FUNCTION_BLOCK A2X_OR_2 (* Composite FB to calculate boolean OR between 2 A2X adapters (UP and DOWN independently) *)
  (* Standard: 61499-2; Function: OUT.UP = IN1.UP OR IN2.UP, OUT.DOWN = IN1.DOWN OR IN2.DOWN; Description: Copyright (c) 2026 HR Agrartechnik GmbH This program and the accompanying materials are made available under the terms of the Eclipse Public License 2.0 which is available at https://www.eclipse.org/legal/epl-2.0/ SPDX-License-Identifier: EPL-2.0 *)
  (* Version 1.0, 2026-08-31, Franz Höpfinger, HR Agrartechnik GmbH, Initial Version *)
  PACKAGE adapter::booleanOperators;
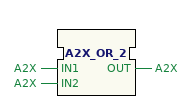
  SOCKETS
    IN1 : adapter::types::unidirectional::A2X; (* OR input 1 *)
    IN2 : adapter::types::unidirectional::A2X; (* OR input 2 *)
  END_SOCKETS
  PLUGS
    OUT : adapter::types::unidirectional::A2X; (* OR result *)
  END_PLUGS
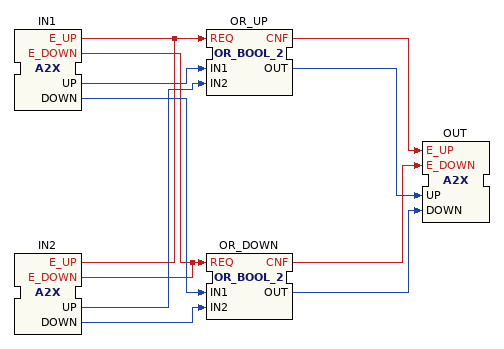
  FBS
    OR_UP : iec61131::booleanOperators::OR_BOOL_2; (* ORs the UP channel *)
    OR_DOWN : iec61131::booleanOperators::OR_BOOL_2; (* ORs the DOWN channel *)
  END_FBS
  EVENT_CONNECTIONS
    IN1.E_UP TO OR_UP.REQ;
    IN2.E_UP TO OR_UP.REQ;
    OR_UP.CNF TO OUT.E_UP;
    IN1.E_DOWN TO OR_DOWN.REQ;
    IN2.E_DOWN TO OR_DOWN.REQ;
    OR_DOWN.CNF TO OUT.E_DOWN;
  END_CONNECTIONS
  DATA_CONNECTIONS
    IN1.UP TO OR_UP.IN1;
    IN2.UP TO OR_UP.IN2;
    OR_UP.OUT TO OUT.UP;
    IN1.DOWN TO OR_DOWN.IN1;
    IN2.DOWN TO OR_DOWN.IN2;
    OR_DOWN.OUT TO OUT.DOWN;
  END_CONNECTIONS
END_FUNCTION_BLOCK
